PROGRAM MAIN
VAR
	
	CountScale : BYTE;

	Mux_Select AT %Q*: ARRAY[0..4] OF BOOL;	
	ADC_Val AT %I* : INT; 
	AnalogRead : ARRAY[0..31] OF INT;
	CLK_MUX : BOOL;
	
	MUX_FUNC : MUX_ADC;

	IO_Out AT %Q* : ARRAY[0..31] OF BOOL;
	IO_In AT %I* : ARRAY[0..16] OF BOOL;
	
	SensAnalaog AT %I* : ARRAY[0..3] OF INT;
	
	RTD_ADC AT %I* : INT;
	RTD_Temp : REAL;
	
	

END_VAR

CLK_MUX := NOT(CLK_MUX);

IO_Out[8] := HMI_Global.HMI_IN_Digital[0];
HMI_Global.HMI_OUT_Analog[0] := AnalogRead[9];

IF AnalogRead[9] > 1000 THEN
	HMI_Global.HMI_OUT_Digital[0] := TRUE;
ELSE
	HMI_Global.HMI_OUT_Digital[0] := FALSE;
END_IF
 

MUX_FUNC(
	CLK := CLK_MUX,
	ADC_INPUT := ADC_Val,
	SELLECT => Mux_Select,
	ADC_OUTPUT => AnalogRead	
);

END_PROGRAM

(* stored: Version 1.1.0.1, ProductVersion 3.1.4024.12
   POU MAIN: Id {57ea5a5e-9fa6-4fd0-90ff-f75dd399de50}, SpecialFunc None *)
